# EPICS autosave request: iocBoot/ioc13MCC/auto_settings.req
file "calc_GSECARS_settings.req",       P=$(P)
file "CARS_motor_settings.req",         P=$(P), M=m1
file "CARS_motor_settings.req",         P=$(P), M=m2
file "CARS_motor_settings.req",         P=$(P), M=m3
